(* CoDeSys 2.3.9.41 project: Котел_розжиг.pro *)
(* Libraries: Standard.lib 4.10.05 11:14:46, SYSLIBCALLBACK.LIB 26.9.08 16:43:52, Util.lib 18.5.10 15:14:28 *)

(* POU PLC_PRG, CFC *)
PROGRAM PLC_PRG
VAR
	valveLowFeed: INT;
	valveGeneralFeed: BOOL;
	valveAlertStop: BOOL;
	tempSensor: BOOL;
	consFuelSensor: INT;
	start: BOOL;
	flameSensor: BOOL;
	igniter: BOOL;
	charCurveVL: CHARCURVE;
	valveIntLV: INT:=20;
	stop: BOOL;
	valveNormalFeed: BOOL;
	trigerIgniter: R_TRIG;
	flameWarning: BOOL;
	tonIgniter: TON;
	rsIgniter: RS;
	trigenIgniterWarning: R_TRIG;
	ctuIgniter: CTU;
	ctusIgniter: INT;
	rsStop: RS;
	vent: INT;
	ventMAX: INT:=20;
	stopVent: BOOL;
	tonVent: TON;
	trigenVentStop: R_TRIG;
	rsStartStop: RS;
	outIgniter: TIME;
	outStopVentTime: TIME;
	rsStopVent: RS;
	fuelSensorLimit: INT:=100;
	valveIndicator: BOOL;
	tpFlameWarning: TP;
	outFlameWarning: TIME;
	tonCtuIgniter: TON;
	outCtuIgniter: TIME;
	stopButton: BOOL;
	rsStopButton: RS;
	startState: BOOL;
	ventWork: BOOL;
	flameButton: BOOL;
	outStopVent: TIME;
	tonStopVent: TON;
	rsStopVentTime: RS;
END_VAR
VAR (* helpers for the ST form of the networks *)
	_t240 : BOOL;
	_t120 : INT;
	_t99 : BOOL;
	_t104 : BOOL;
	_t34 : BOOL;
	_t187 : BOOL;
	_t61 : INT;
	_t56 : BOOL;
	_t16 : BOOL;
	_t110 : BOOL;
	_t29 : BOOL;
	_t31 : BOOL;
	_t89 : BOOL;
	_t51 : INT;
	_t50 : INT;
	_t112 : BOOL;
	_t208 : BOOL;
	_t133 : BOOL;
	_t121 : BOOL;
END_VAR
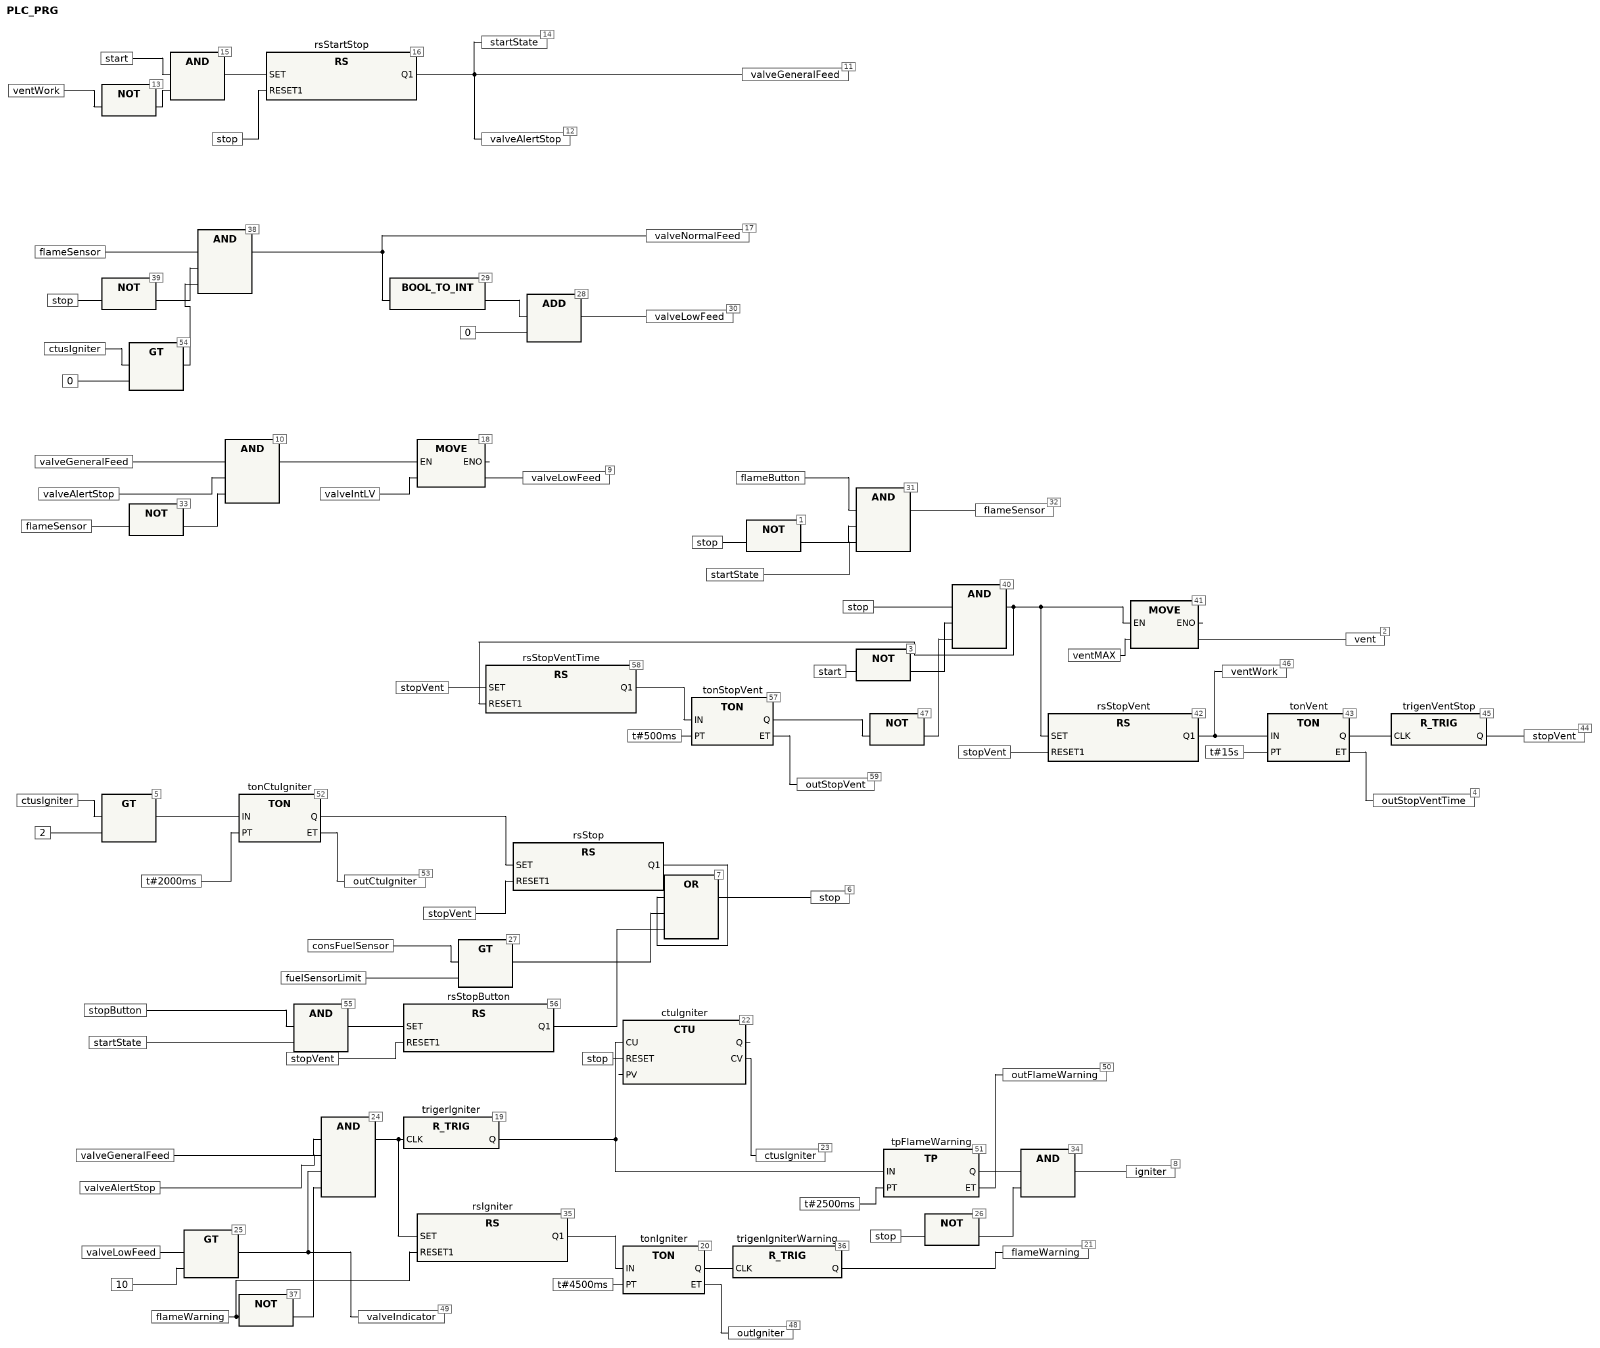
_CFC_ (* Continuous Function Chart, elements in execution order *)
#0 rsStop:RS(SET: #52.Q, RESET1: stopVent)
#1 NOT(stop)
#2 vent <= #41
#3 NOT(start)
#4 outStopVentTime <= #43.ET
#5 GT(ctusIgniter, 2)
#6 stop <= #7
#7 OR(#0.Q1, #27, #56.Q1)
#8 igniter <= #34
#9 valveLowFeed <= #18
#10 AND(valveGeneralFeed, valveAlertStop, #33)
#11 valveGeneralFeed <= #16.Q1
#12 valveAlertStop <= #16.Q1
#13 NOT(ventWork)
#14 startState <= #16.Q1
#15 AND(start, #13)
#16 rsStartStop:RS(SET: #15, RESET1: stop)
#17 valveNormalFeed <= #38
#18 MOVE(EN: #10, valveIntLV)
#19 trigerIgniter:R_TRIG(CLK: #24)
#20 tonIgniter:TON(IN: #35.Q1, PT: t#4500ms)
#21 flameWarning <= #36.Q
#22 ctuIgniter:CTU(CU: #19.Q, RESET: stop, PV: -)
#23 ctusIgniter <= #22.CV
#24 AND(valveGeneralFeed, valveAlertStop, #25, #37)
#25 GT(valveLowFeed, 10)
#26 NOT(stop)
#27 GT(consFuelSensor, fuelSensorLimit)
#28 ADD(#29, 0)
#29 BOOL_TO_INT(#38)
#30 valveLowFeed <= #28
#31 AND(flameButton, #1, startState)
#32 flameSensor <= #31
#33 NOT(flameSensor)
#34 AND(#51.Q, #26)
#35 rsIgniter:RS(SET: #24, RESET1: flameWarning)
#36 trigenIgniterWarning:R_TRIG(CLK: #20.Q)
#37 NOT(flameWarning)
#38 AND(flameSensor, #39, #54)
#39 NOT(stop)
#40 AND(stop, #3, #47)
#41 MOVE(EN: #40, ventMAX)
#42 rsStopVent:RS(SET: #40, RESET1: stopVent)
#43 tonVent:TON(IN: #42.Q1, PT: t#15s)
#44 stopVent <= #45.Q
#45 trigenVentStop:R_TRIG(CLK: #43.Q)
#46 ventWork <= #42.Q1
#47 NOT(#57.Q)
#48 outIgniter <= #20.ET
#49 valveIndicator <= #25
#50 outFlameWarning <= #51.ET
#51 tpFlameWarning:TP(IN: #19.Q, PT: t#2500ms)
#52 tonCtuIgniter:TON(IN: #5, PT: t#2000ms)
#53 outCtuIgniter <= #52.ET
#54 GT(ctusIgniter, 0)
#55 AND(stopButton, startState)
#56 rsStopButton:RS(SET: #55, RESET1: stopVent)
#57 tonStopVent:TON(IN: #58.Q1, PT: t#500ms)
#58 rsStopVentTime:RS(SET: stopVent, RESET1: #40)
#59 outStopVent <= #57.ET
_END_CFC_
(* the same logic as Structured Text *)
rsStop(SET := tonCtuIgniter.Q, RESET1 := stopVent);
_t240 := NOT stop;
vent := _t120;
outStopVentTime := tonVent.ET;
_t99 := ctusIgniter > 2;
stop := _t104;
_t104 := rsStop.Q1 OR _t34 OR rsStopButton.Q1;
igniter := _t187;
valveLowFeed := _t61;
_t16 := valveGeneralFeed AND valveAlertStop AND _t56;
valveGeneralFeed := rsStartStop.Q1;
valveAlertStop := rsStartStop.Q1;
startState := rsStartStop.Q1;
rsStartStop(SET := start AND NOT ventWork, RESET1 := stop);
valveNormalFeed := _t110;
IF _t16 THEN _t61 := valveIntLV; END_IF;
trigerIgniter(CLK := _t29);
tonIgniter(IN := rsIgniter.Q1, PT := t#4500ms);
flameWarning := trigenIgniterWarning.Q;
ctuIgniter(CU := trigerIgniter.Q, RESET := stop);
ctusIgniter := ctuIgniter.CV;
_t29 := valveGeneralFeed AND valveAlertStop AND _t31 AND _t89;
_t31 := valveLowFeed > 10;
_t34 := consFuelSensor > fuelSensorLimit;
_t50 := _t51 + 0;
_t51 := BOOL_TO_INT(_t110);
valveLowFeed := _t50;
flameSensor := flameButton AND _t240 AND startState;
_t56 := NOT flameSensor;
_t187 := tpFlameWarning.Q AND NOT stop;
rsIgniter(SET := _t29, RESET1 := flameWarning);
trigenIgniterWarning(CLK := tonIgniter.Q);
_t89 := NOT flameWarning;
_t110 := flameSensor AND _t112 AND _t208;
_t112 := NOT stop;
_t121 := stop AND NOT start AND _t133;
IF _t121 THEN _t120 := ventMAX; END_IF;
rsStopVent(SET := _t121, RESET1 := stopVent);
tonVent(IN := rsStopVent.Q1, PT := t#15s);
stopVent := trigenVentStop.Q;
trigenVentStop(CLK := tonVent.Q);
ventWork := rsStopVent.Q1;
_t133 := NOT tonStopVent.Q;
outIgniter := tonIgniter.ET;
valveIndicator := _t31;
outFlameWarning := tpFlameWarning.ET;
tpFlameWarning(IN := trigerIgniter.Q, PT := t#2500ms);
tonCtuIgniter(IN := _t99, PT := t#2000ms);
outCtuIgniter := tonCtuIgniter.ET;
_t208 := ctusIgniter > 0;
rsStopButton(SET := stopButton AND startState, RESET1 := stopVent);
tonStopVent(IN := rsStopVentTime.Q1, PT := t#500ms);
rsStopVentTime(SET := stopVent, RESET1 := _t121);
outStopVent := tonStopVent.ET;
END_PROGRAM

(* Visualisation ignition
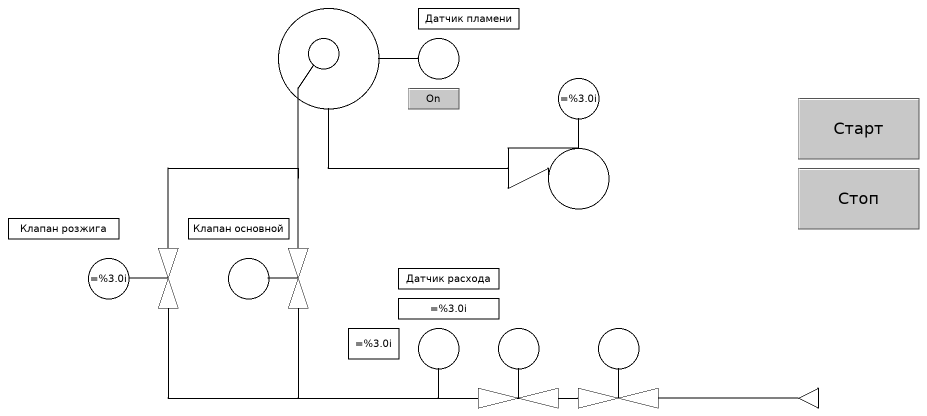
ellipse at (330,300)-(371,341): alarm colour if PLC_PRG.valveNormalFeed
ellipse at (190,300)-(231,341): text "=%3.0i"; shows PLC_PRG.valveLowFeed; alarm colour if PLC_PRG.valveIndicator; editable 0..100
ellipse at (410,80)-(441,111): alarm colour if PLC_PRG.igniter
ellipse at (520,80)-(561,121): alarm colour if PLC_PRG.flameSensor
ellipse at (700,370)-(741,411): alarm colour if PLC_PRG.valveGeneralFeed
rectangle at (520,50)-(621,71): text "Датчик пламени"
rectangle at (500,310)-(601,331): text "Датчик расхода"
rectangle at (110,260)-(221,281): text "Клапан розжига"
rectangle at (290,260)-(391,281): text "Клапан основной"
button at (900,140)-(1021,201): text "Старт"; taps PLC_PRG.start
button at (900,210)-(1021,271): text "Стоп"; taps PLC_PRG.stopButton
ellipse at (660,120)-(701,161): text "=%3.0i"; shows PLC_PRG.vent; alarm colour if PLC_PRG.ventWork
button at (510,130)-(561,151): text "On"; toggles PLC_PRG.flameButton
rectangle at (500,340)-(601,361): text "=%3.0i"; shows PLC_PRG.fuelSensorLimit; editable 0..1000
rectangle at (450,370)-(501,401): text "=%3.0i"; shows PLC_PRG.consFuelSensor; editable 0..1000
ellipse at (600,370)-(641,411): alarm colour if PLC_PRG.valveAlertStop
22 more shapes without text or variables
*)
